TYPE ST_MachineParametersAxis :
STRUCT
	fSoftPositionLimitMax			: LREAL;
	fSoftPositionLimitMin			: LREAL;
	fDefaultVelocity				: LREAL;
	fHomePosition					: LREAL;
END_STRUCT
END_TYPE

(* stored: Version 1.1.0.1, ProductVersion 3.1.4024.11
   DUT ST_MachineParametersAxis: Id {116e8143-6223-4ba3-b095-925f46ea32c4} *)
